ABB RAPID module: Module1.mod

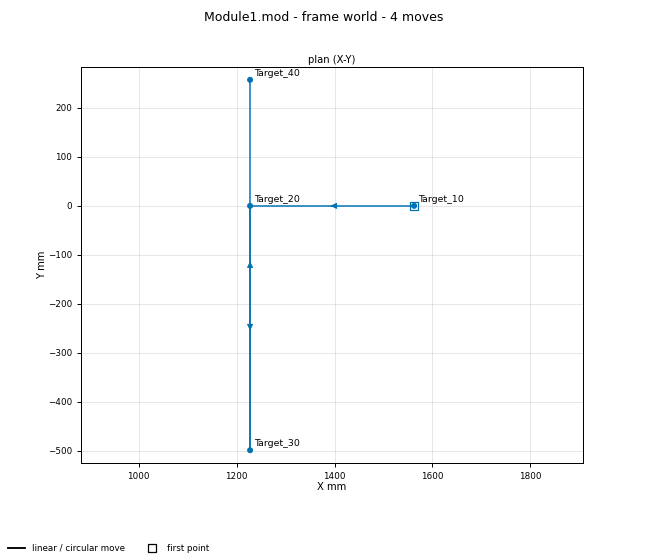
[picture p0: tool path of Module1.mod in frame world, 4 of 4 moves have a stored position in this frame; points joined in program order, loops and branches not executed]
MODULE Module1
    CONST robtarget Target_10:=[[1562.5,0,1931.794919243],[0.258819045,0,0.965925826,0],[0,0,0,0],[0,9E+09,9E+09,9E+09,9E+09,9E+09]];
    CONST robtarget Target_20:=[[1227.413978312,0,1931.795026584],[0.258819017,0,0.965925834,0],[0,0,0,0],[0,9E+09,9E+09,9E+09,9E+09,9E+09]];
    CONST robtarget Target_30:=[[1227.413991094,-499.175760145,1931.795029505],[0.258819029,-0.000000007,0.965925831,-0.000000001],[-1,0,-1,0],[0,9E+09,9E+09,9E+09,9E+09,9E+09]];
    CONST robtarget Target_40:=[[1227.414000588,257.42908943,1931.795015248],[0.258819039,-0.000000015,0.965925828,0.000000001],[0,-1,0,0],[0,9E+09,9E+09,9E+09,9E+09,9E+09]];
    PROC Path_10()
        MoveJ Target_10,v100,z100,tool0\WObj:=wobj0;
        MoveL Target_20,v100,z100,tool0\WObj:=wobj0;
        MoveL Target_30,v100,z100,tool0\WObj:=wobj0;
        MoveL Target_40,v100,z100,tool0\WObj:=wobj0;
    ENDPROC
ENDMODULE
